FUNCTION_BLOCK TEST_NE2 (* Test "<>" in ECC transition *)
  (* Standard: 61499-2 *)
  (* Version 0.0, 2002-12-17, JHC, Rockwell Automation *)
  (* Compiler header: package fb.rt.test; *)
  (* Compiler Java IBM JIkes 1.06 *)
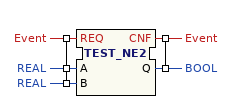
  EVENT_INPUT
    REQ WITH A, B; (* Normal Execution Request *)
  END_EVENT
  EVENT_OUTPUT
    CNF WITH Q; (* Execution Confirmation *)
  END_EVENT
  VAR_INPUT
    A : REAL;
    B : REAL;
  END_VAR
  VAR_OUTPUT
    Q : BOOL; (* A <> B? *)
  END_VAR
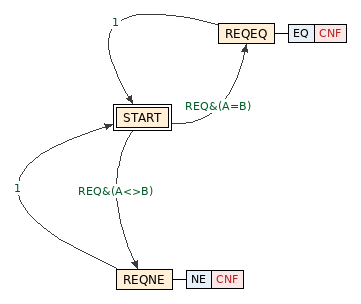
  EC_STATES
    START; (* Initial State *)
    REQEQ : EQ -> CNF; (* Execution when A=B *)
    REQNE : NE -> CNF; (* Execution when A<>B *)
  END_STATES
  EC_TRANSITIONS
    START TO REQEQ := REQ&(A=B);
    START TO REQNE := REQ&(A<>B);
    REQEQ TO START := 1;
    REQNE TO START := 1;
  END_TRANSITIONS
  ALGORITHM EQ IN ST: (* Algorithm when A=B *)
Q := FALSE;
  END_ALGORITHM
  ALGORITHM NE IN ST: (* Algorithm when A<>B *)
Q := TRUE;
  END_ALGORITHM
END_FUNCTION_BLOCK
